(* IEC 61131-3 sources: ics/BLR101_ProenixContact/BLR101_5_ILC171_44/LogicalPOUs/AIO, 3 files *)

(* ---- SensorFB.ST ---- *)
(*@PROPERTIES_EX@
TYPE: POU
LOCALE: 0
IEC_LANGUAGE: ST
PLC_TYPE: independent
PROC_TYPE: independent
GROUP: AIO.FB
*)
(*@KEY@:DESCRIPTION*)

(*@KEY@:END_DESCRIPTION*)
FUNCTION_BLOCK SensorFB

(*Group:Default*)

VAR_IN_OUT
	Snsr_strct :	SNSR;
END_VAR

VAR
	RealValue :	REAL;
	bar_kgf :	REAL;
END_VAR

VAR_IN_OUT
	Buff :	SNSR_BUFF;
END_VAR

VAR
	SumValue :	REAL;
	y :	INT;
	INIT :	BOOL;
	FltrValue :	REAL;
	x :	INT;
END_VAR

VAR_OUTPUT
	Event :	SNSR_EVENT;
END_VAR

VAR_IN_OUT
	Aux_strct :	SNSR_MISC;
END_VAR

VAR_EXTERNAL
	TICK_100MS_PLS :	BOOL;
END_VAR

(*@KEY@: WORKSHEET
NAME: SensorFB
IEC_LANGUAGE: ST
*)

(*================================================================================================*)
(*Fault operation & converting PIW to real value*)
(*================================================================================================*)
IF (Snsr_strct.PIW < 0) OR (Snsr_strct.PIW > Snsr_strct.ADC_Range) OR Snsr_strct.CW.ExtFault OR (Snsr_strct.DiagCode > word#16#8000) THEN		(*Snsr_strct Failed*)
	Snsr_strct.SW.Fault:= TRUE;
	RealValue:= 0.0;
ELSE                                                                    			(*Snsr_strct OK*)
	IF Snsr_strct.ADC_Range <= 0 THEN
		Snsr_strct.ADC_Range:= 1;
	END_IF;
	Snsr_strct.SW.Fault:= FALSE;
	RealValue:= (Snsr_strct.Ymax - Snsr_strct.Ymin) * bar_kgf * INT_TO_REAL(Snsr_strct.PIW) / INT_TO_REAL(Snsr_strct.ADC_Range) + Snsr_strct.Ymin ;
END_IF;

(*================================================================================================*)
(*Converting from bar to kgf/sm2*)
(*================================================================================================*)
IF Snsr_strct.CW.bar_kgf THEN
	bar_kgf:= 1.0197;
ELSE
	bar_kgf:= 1.0;
END_IF;

(*================================================================================================*)
(*SMA filter operation*)
(*================================================================================================*)
if INIT then
	if TICK_100MS_PLS then
		Aux_strct.SamplingTickCount:= Aux_strct.SamplingTickCount + 1;
	end_if;
else
	Aux_strct.SamplingTickCount:= 0;
end_if;

IF Snsr_strct.CW.FltrEn THEN
	IF NOT INIT THEN																(*Initialization*)
		FOR y:= 0 TO 9 DO
			Buff[y]:= RealValue;
			SumValue:= SumValue + Buff[y];
		END_FOR;
		INIT:= TRUE;
	ELSE
		IF Aux_strct.SamplingTickCount >= (Snsr_strct.SamplingTime * 10) THEN		(*Buffer shifting and changing last element*)
			FOR y:= 0 TO 8 DO
				x:= y + 1;
				Buff[y]:= Buff[x];
			END_FOR;
			Buff[9]:= RealValue;
			SumValue:= SumValue + RealValue - Buff[0];
			Aux_strct.SamplingTickCount:= 0;
		END_IF;
		FltrValue:= SumValue / 10.0;
	END_IF;
ELSE
	INIT:= FALSE;
	SumValue:= 0.0;
	FltrValue:= 0.0;
END_IF;

(*================================================================================================*)
(*Snsr_strct output values states*)
(*================================================================================================*)
IF Snsr_strct.CW.SimEn THEN															(*Simulated output value*)
	Snsr_strct.RealValue:= Snsr_strct.SimValue;
ELSIF Snsr_strct.CW.FltrEn THEN														(*Filtered output value*)
	Snsr_strct.RealValue:= FltrValue;
ELSE																				(*Real output value*)
	Snsr_strct.RealValue:= RealValue;
END_IF;

Snsr_strct.IntValue:= REAL_TO_INT(Snsr_strct.RealValue * 100.0);

(*================================================================================================*)
(*Limits operation*)
(*================================================================================================*)
if Snsr_strct.CW.LimEn then
	if (Snsr_strct.RealValue > (Snsr_strct.HH + (Snsr_strct.DeadBand / 2.0))) and not Snsr_strct.SW.HH_alarm  then
		if TICK_100MS_PLS then
			Aux_strct.HHTopDelayCount:= Aux_strct.HHTopDelayCount + 1;
		end_if;
		if Aux_strct.HHTopDelayCount > (Snsr_strct.LimDelay * 10) then
			Snsr_strct.SW.HH_alarm:= true;
		end_if;
	else
		Aux_strct.HHTopDelayCount:= 0;
	end_if;

	if (Snsr_strct.RealValue < (Snsr_strct.HH - (Snsr_strct.DeadBand / 2.0))) and Snsr_strct.SW.HH_alarm then
		if TICK_100MS_PLS then
			Aux_strct.HHBotDelayCount:= Aux_strct.HHBotDelayCount + 1;
		end_if;
		if Aux_strct.HHBotDelayCount > (Snsr_strct.LimDelay * 10) then
			Snsr_strct.SW.HH_alarm:= false;
		end_if;
	else
		Aux_strct.HHBotDelayCount:= 0;
	end_if;

	if (Snsr_strct.RealValue > (Snsr_strct.HL + (Snsr_strct.DeadBand / 2.0))) and not Snsr_strct.SW.HL_alarm then
		if TICK_100MS_PLS then
			Aux_strct.HLTopDelayCount:= Aux_strct.HLTopDelayCount + 1;
		end_if;
		if Aux_strct.HLTopDelayCount > (Snsr_strct.LimDelay * 10) then
			Snsr_strct.SW.HL_alarm:= true;
		end_if;
	else
		Aux_strct.HLTopDelayCount:= 0;
	end_if;

	if (Snsr_strct.RealValue < (Snsr_strct.HL - (Snsr_strct.DeadBand / 2.0))) and Snsr_strct.SW.HL_alarm then
		if TICK_100MS_PLS then
			Aux_strct.HLBotDelayCount:= Aux_strct.HLBotDelayCount + 1;
		end_if;
		if Aux_strct.HLBotDelayCount > (Snsr_strct.LimDelay * 10) then
			Snsr_strct.SW.HL_alarm:= false;
		end_if;
	else
		Aux_strct.HLBotDelayCount:= 0;
	end_if;

	if (Snsr_strct.RealValue < (Snsr_strct.LH - (Snsr_strct.DeadBand / 2.0))) and not Snsr_strct.SW.LH_alarm then
		if TICK_100MS_PLS then
			Aux_strct.LHTopDelayCount:= Aux_strct.LHTopDelayCount + 1;
		end_if;
		if Aux_strct.LHTopDelayCount > (Snsr_strct.LimDelay * 10) then
			Snsr_strct.SW.LH_alarm:= true;
		end_if;
	else
		Aux_strct.LHTopDelayCount:= 0;
	end_if;

	if (Snsr_strct.RealValue > (Snsr_strct.LH + (Snsr_strct.DeadBand / 2.0))) and Snsr_strct.SW.LH_alarm then
		if TICK_100MS_PLS then
			Aux_strct.LHBotDelayCount:= Aux_strct.LHBotDelayCount + 1;
		end_if;
		if Aux_strct.LHBotDelayCount > (Snsr_strct.LimDelay * 10) then
			Snsr_strct.SW.LH_alarm:= false;
		end_if;
	else
		Aux_strct.LHBotDelayCount:= 0;
	end_if;

	if (Snsr_strct.RealValue < (Snsr_strct.LL - (Snsr_strct.DeadBand / 2.0))) and not Snsr_strct.SW.LL_alarm then
		if TICK_100MS_PLS then
			Aux_strct.LLTopDelayCount:= Aux_strct.LLTopDelayCount + 1;
		end_if;
		if Aux_strct.LLTopDelayCount > (Snsr_strct.LimDelay * 10) then
			Snsr_strct.SW.LL_alarm:= true;
		end_if;
	else
		Aux_strct.LLTopDelayCount:= 0;
	end_if;

	if (Snsr_strct.RealValue > (Snsr_strct.LL + (Snsr_strct.DeadBand / 2.0))) and Snsr_strct.SW.LL_alarm then
		if TICK_100MS_PLS then
			Aux_strct.LLBotDelayCount:= Aux_strct.LLBotDelayCount + 1;
		end_if;
		if Aux_strct.LLBotDelayCount > (Snsr_strct.LimDelay * 10) then
			Snsr_strct.SW.LL_alarm:= false;
		end_if;
	else
		Aux_strct.LLBotDelayCount:= 0;
	end_if;

else
	Aux_strct.HHTopDelayCount:= 0;
	Aux_strct.HHBotDelayCount:= 0;

	Aux_strct.HLTopDelayCount:= 0;
	Aux_strct.HLBotDelayCount:= 0;

	Aux_strct.LHTopDelayCount:= 0;
	Aux_strct.LHBotDelayCount:= 0;

	Aux_strct.LLTopDelayCount:= 0;
	Aux_strct.LLBotDelayCount:= 0;

	Snsr_strct.SW.HH_alarm:= FALSE;
	Snsr_strct.SW.HL_alarm:= FALSE;
	Snsr_strct.SW.LH_alarm:= FALSE;
	Snsr_strct.SW.LL_alarm:= FALSE;
end_if;

(*================================================================================================*)
(*Sensor Pulse Events*)
(*================================================================================================*)

Event.Fault:= false;
if Snsr_strct.SW.Fault and not Aux_strct.EVENT_1 then
	Event.Fault:= true;
	Aux_strct.EVENT_1:= true;
elsif not Snsr_strct.SW.Fault then
	Aux_strct.EVENT_1:= false;
end_if;

Event.HH:= false;
if Snsr_strct.SW.HH_alarm and not Aux_strct.EVENT_2 then
	Event.HH:= true;
	Aux_strct.EVENT_2:= true;
elsif not Snsr_strct.SW.HH_alarm then
	Aux_strct.EVENT_2:= false;
end_if;

Event.HL:= false;
if Snsr_strct.SW.HL_alarm and not Aux_strct.EVENT_3 then
	Event.HL:= true;
	Aux_strct.EVENT_3:= true;
elsif not Snsr_strct.SW.HL_alarm then
	Aux_strct.EVENT_3:= false;
end_if;

Event.LH:= false;
if Snsr_strct.SW.LH_alarm and not Aux_strct.EVENT_4 then
	Event.LH:= true;
	Aux_strct.EVENT_4:= true;
elsif not Snsr_strct.SW.LH_alarm then
	Aux_strct.EVENT_4:= false;
end_if;

Event.LL:= false;
if Snsr_strct.SW.LL_alarm and not Aux_strct.EVENT_5 then
	Event.LL:= true;
	Aux_strct.EVENT_5:= true;
elsif not Snsr_strct.SW.LL_alarm then
	Aux_strct.EVENT_5:= false;
end_if;

(*@KEY@: END_WORKSHEET *)
END_FUNCTION_BLOCK

(* ---- AI.ST ---- *)
(*@PROPERTIES_EX@
TYPE: POU
LOCALE: 0
IEC_LANGUAGE: ST
PLC_TYPE: independent
PROC_TYPE: independent
GROUP: AIO
*)
(*@KEY@:DESCRIPTION*)

(*@KEY@:END_DESCRIPTION*)
PROGRAM AI

(*Group:Default*)

VAR_EXTERNAL
	AI :	SENSOR;
END_VAR

VAR
	A07_Param :	IL_AI_4_UI_Para_V1_03;
	i :	INT;
	j :	INT;
	udtA07Param :	ANL_udt_Para_1_5;
	A07_Com :	IL_AI_4_UI_Com_V1_04;
	udtA07Status :	ANL_udt_Status_1_5;
	A07_Ready :	BOOL;
	A07_Err :	BOOL;
	A07_Frmwr :	STRING;
END_VAR

VAR_EXTERNAL
	A07_ProcIn :	ANL_ARR_W_1_4;
	A07_ProcOut :	ANL_ARR_W_1_4;
END_VAR

VAR
	A07_DiagCode :	WORD;
	A07_Diag :	IL_AI_4_UI_Diag_V1_03;
	A08_Param :	IL_AI_4_UI_Para_V1_03;
	udtA08Param :	ANL_udt_Para_1_5;
	A08_Com :	IL_AI_4_UI_Com_V1_04;
	A08_Ready :	BOOL;
	A08_Err :	BOOL;
	A08_DiagCode :	WORD;
	A08_Frmwr :	STRING;
	udtA08Status :	ANL_udt_Status_1_5;
END_VAR

VAR_EXTERNAL
	A08_ProcIn :	ANL_ARR_W_1_4;
	A08_ProcOut :	ANL_ARR_W_1_4;
END_VAR

VAR
	A08_Diag :	IL_AI_4_UI_Diag_V1_03;
	A09_Param :	IL_AI_4_UI_Para_V1_03;
	udtA09Param :	ANL_udt_Para_1_5;
	A09_Com :	IL_AI_4_UI_Com_V1_04;
	A09_Ready :	BOOL;
	A09_Err :	BOOL;
	A09_DiagCode :	WORD;
	A09_Frmwr :	STRING;
	udtA09Status :	ANL_udt_Status_1_5;
END_VAR

VAR_EXTERNAL
	A09_ProcIn :	ANL_ARR_W_1_4;
	A09_ProcOut :	ANL_ARR_W_1_4;
END_VAR

VAR
	A09_Diag :	IL_AI_4_UI_Diag_V1_03;
	A10_Param :	IL_AI_4_UI_Para_V1_03;
	udtA10Param :	ANL_udt_Para_1_5;
	A10_Com :	IL_AI_4_UI_Com_V1_04;
	A10_Ready :	BOOL;
	A10_Err :	BOOL;
	A10_Frmwr :	STRING;
	udtA10Status :	ANL_udt_Status_1_5;
END_VAR

VAR_EXTERNAL
	A10_ProcIn :	ANL_ARR_W_1_4;
	A10_ProcOut :	ANL_ARR_W_1_4;
END_VAR

VAR
	A10_Diag :	IL_AI_4_UI_Diag_V1_03;
	A11_Param :	IL_AI_4_UI_Para_V1_03;
	udtA11Param :	ANL_udt_Para_1_5;
	A11_Com :	IL_AI_4_UI_Com_V1_04;
	A11_Ready :	BOOL;
	A11_Err :	BOOL;
	A11_DiagCode :	WORD;
	A11_Frmwr :	STRING;
	udtA11Status :	ANL_udt_Status_1_5;
END_VAR

VAR_EXTERNAL
	A11_ProcIn :	ANL_ARR_W_1_4;
	A11_ProcOut :	ANL_ARR_W_1_4;
END_VAR

VAR
	A11_Diag :	IL_AI_4_UI_Diag_V1_03;
	A10_DiagCode :	WORD;
	A12_Param :	IL_AI_4_UI_Para_V1_03;
	udtA12Param :	ANL_udt_Para_1_5;
	A12_Com :	IL_AI_4_UI_Com_V1_04;
	A12_Ready :	BOOL;
	A12_Err :	BOOL;
	A12_DiagCode :	WORD;
	A12_Frmwr :	STRING;
	udtA12Status :	ANL_udt_Status_1_5;
END_VAR

VAR_EXTERNAL
	A12_ProcIn :	ANL_ARR_W_1_4;
	A12_ProcOut :	ANL_ARR_W_1_4;
END_VAR

VAR
	A12_Diag :	IL_AI_4_UI_Diag_V1_03;
	SensorsFB :	SensorFB;
	AI_BUFF :	SENSOR_BUFF;
END_VAR

VAR_EXTERNAL
	AI_AUX :	SENSOR_MISC;
	AI_EVENT :	SENSOR_EVENT;
END_VAR

VAR
	A07_Param_2 :	IL_AI_4_UI_Para_V1_03;
	A07_Param_3 :	IL_AI_4_UI_Para_V1_03;
	A07_Param_4 :	IL_AI_4_UI_Para_V1_03;
	REAL_TO_MB :	REAL_TO_MB;
	j1 :	INT;
END_VAR

VAR_EXTERNAL
	MBTCP_Data :	MB_TCP_ARR_W_0_7167;
END_VAR

VAR
	j2 :	INT;
END_VAR

(*@KEY@: WORKSHEET
NAME: AI
IEC_LANGUAGE: ST
*)

(*========================================================================================*)
	(*A07 module parametrization*)
(*========================================================================================*)
for i:= 1 to 4 do
	j:= i - 1;
	A07_Param(iChannel:= i,iMode:= 1,iFilter:= 0,rHighLimit:= int_to_real(AI[j].ADC_Range),rLowLimit:= 0.0,udtPara:= udtA07Param);
	udtA07Param:= A07_Param.udtPara;
end_for;

(*========================================================================================*)
	(*A07 module communication*)
(*========================================================================================*)
A07_Com(xActivate:= true,bSelect:= byte#16#0F,xVoltage:= false,udtPara:=udtA07Param,arrProcIn:= A07_ProcIn);
	A07_Ready			:=	A07_Com.xReady;
	A07_Err				:=	A07_Com.xError;
	A07_DiagCode		:=	A07_Com.wDiagCode;
	A07_Frmwr			:=	A07_Com.strFirmware;
	udtA07Status		:=	A07_Com.udtStatus;
	udtA07Param 		:=	A07_Com.udtPara;
	A07_ProcOut			:=	A07_Com.arrProcOut;
(*========================================================================================*)
	(*A07 module diagnostic*)
(*========================================================================================*)
for i:= 1 to 4 do
	j:= i - 1;
	A07_Diag(udtStatus:= udtA07Status,iChannel:= i);
	AI[j].CW.ExtFault:= not A07_Diag.xDataValid;
	AI[j].DiagCode:= A07_Diag.wDiagCode;
	AI[j].PIW:= real_to_int(A07_Diag.rCurrentValue);
end_for;

(*========================================================================================*)
	(*A08 module parametrization*)
(*========================================================================================*)
for i:= 1 to 4 do
	j:= i + 3;
	A08_Param(iChannel:= i,iMode:= 1,iFilter:= 0,rHighLimit:= int_to_real(AI[j].ADC_Range),rLowLimit:= 0.0,udtPara:= udtA08Param);
	udtA08Param:= A08_Param.udtPara;
end_for;

(*========================================================================================*)
	(*A08 module communication*)
(*========================================================================================*)
A08_Com(xActivate:= true,bSelect:= byte#16#0F,xVoltage:= false,udtPara:=udtA08Param,arrProcIn:= A08_ProcIn);
	A08_Ready			:=	A08_Com.xReady;
	A08_Err				:=	A08_Com.xError;
	A08_DiagCode		:=	A08_Com.wDiagCode;
	A08_Frmwr			:=	A08_Com.strFirmware;
	udtA08Status		:=	A08_Com.udtStatus;
	udtA08Param 		:=	A08_Com.udtPara;
	A08_ProcOut			:=	A08_Com.arrProcOut;
(*========================================================================================*)
	(*A08 module diagnostic*)
(*========================================================================================*)
for i:= 1 to 4 do
	j:= i + 3;
	A08_Diag(udtStatus:= udtA08Status,iChannel:= i);
	AI[j].CW.ExtFault:= not A08_Diag.xDataValid;
	AI[j].DiagCode:= A08_Diag.wDiagCode;
	AI[j].PIW:= real_to_int(A08_Diag.rCurrentValue);
end_for;

(*========================================================================================*)
	(*A09 module parametrization*)
(*========================================================================================*)
for i:= 1 to 4 do
	j:= i + 7;
	A09_Param(iChannel:= i,iMode:= 1,iFilter:= 0,rHighLimit:= int_to_real(AI[j].ADC_Range),rLowLimit:= 0.0,udtPara:= udtA09Param);
	udtA09Param:= A09_Param.udtPara;
end_for;

(*========================================================================================*)
	(*A09 module communication*)
(*========================================================================================*)
A09_Com(xActivate:= true,bSelect:= byte#16#0F,xVoltage:= false,udtPara:=udtA09Param,arrProcIn:= A09_ProcIn);
	A09_Ready			:=	A09_Com.xReady;
	A09_Err				:=	A09_Com.xError;
	A09_DiagCode		:=	A09_Com.wDiagCode;
	A09_Frmwr			:=	A09_Com.strFirmware;
	udtA09Status		:=	A09_Com.udtStatus;
	udtA09Param 		:=	A09_Com.udtPara;
	A09_ProcOut			:=	A09_Com.arrProcOut;
(*========================================================================================*)
	(*A09 module diagnostic*)
(*========================================================================================*)
for i:= 1 to 4 do
	j:= i + 7;
	A09_Diag(udtStatus:= udtA09Status,iChannel:= i);
	AI[j].CW.ExtFault:= not A09_Diag.xDataValid;
	AI[j].DiagCode:= A09_Diag.wDiagCode;
	AI[j].PIW:= real_to_int(A09_Diag.rCurrentValue);
end_for;

(*========================================================================================*)
	(*A10 module parametrization*)
(*========================================================================================*)
	A10_Param(iChannel:= 1,iMode:= 1,iFilter:= 0,rHighLimit:= int_to_real(AI[12].ADC_Range),rLowLimit:= 0.0,udtPara:= udtA10Param);
	udtA10Param:= A10_Param.udtPara;

(*========================================================================================*)
	(*A10 module communication*)
(*========================================================================================*)
A10_Com(xActivate:= true,bSelect:= byte#16#01,xVoltage:= false,udtPara:=udtA10Param,arrProcIn:= A10_ProcIn);
	A10_Ready			:=	A10_Com.xReady;
	A10_Err				:=	A10_Com.xError;
	A10_DiagCode		:=	A10_Com.wDiagCode;
	A10_Frmwr			:=	A10_Com.strFirmware;
	udtA10Status		:=	A10_Com.udtStatus;
	udtA10Param 		:=	A10_Com.udtPara;
	A10_ProcOut			:=	A10_Com.arrProcOut;
(*========================================================================================*)
	(*A10 module diagnostic*)
(*========================================================================================*)
	A10_Diag(udtStatus:= udtA10Status,iChannel:= 1);
	AI[12].CW.ExtFault:= not A10_Diag.xDataValid;
	AI[12].DiagCode:= A10_Diag.wDiagCode;
	AI[12].PIW:= real_to_int(A10_Diag.rCurrentValue);

(*========================================================================================*)
	(*A11 module parametrization*)
(*========================================================================================*)
for i:= 1 to 3 do
	j:= i + 15;
	A11_Param(iChannel:= i,iMode:= 0,iFilter:= 0,rHighLimit:= 10000.0,rLowLimit:= 0.0,udtPara:= udtA11Param);
	udtA11Param:= A11_Param.udtPara;
end_for;

(*========================================================================================*)
	(*A11 module communication*)
(*========================================================================================*)
A11_Com(xActivate:= true,bSelect:= byte#16#07,xVoltage:= false,udtPara:=udtA11Param,arrProcIn:= A11_ProcIn);
	A11_Ready			:=	A11_Com.xReady;
	A11_Err				:=	A11_Com.xError;
	A11_DiagCode		:=	A11_Com.wDiagCode;
	A11_Frmwr			:=	A11_Com.strFirmware;
	udtA11Status		:=	A11_Com.udtStatus;
	udtA11Param 		:=	A11_Com.udtPara;
	A11_ProcOut			:=	A11_Com.arrProcOut;
(*========================================================================================*)
	(*A11 module diagnostic*)
(*========================================================================================*)
for i:= 1 to 3 do
	j:= i + 15;
	A11_Diag(udtStatus:= udtA11Status,iChannel:= i);
	AI[j].CW.ExtFault:= not A11_Diag.xDataValid;
	AI[j].DiagCode:= A11_Diag.wDiagCode;
	AI[j].PIW:= real_to_int(A11_Diag.rCurrentValue);
end_for;

(*========================================================================================*)
	(*A12 module parametrization*)
(*========================================================================================*)
for i:= 1 to 2 do
	j:= i + 19;
	A12_Param(iChannel:= i,iMode:= 0,iFilter:= 0,rHighLimit:= 10000.0,rLowLimit:= 0.0,udtPara:= udtA12Param);
	udtA12Param:= A12_Param.udtPara;
end_for;

(*========================================================================================*)
	(*A12 module communication*)
(*========================================================================================*)
A12_Com(xActivate:= true,bSelect:= byte#16#03,xVoltage:= false,udtPara:=udtA12Param,arrProcIn:= A12_ProcIn);
	A12_Ready			:=	A12_Com.xReady;
	A12_Err				:=	A12_Com.xError;
	A12_DiagCode		:=	A12_Com.wDiagCode;
	A12_Frmwr			:=	A12_Com.strFirmware;
	udtA12Status		:=	A12_Com.udtStatus;
	udtA12Param 		:=	A12_Com.udtPara;
	A12_ProcOut			:=	A12_Com.arrProcOut;
(*========================================================================================*)
	(*A12 module diagnostic*)
(*========================================================================================*)
for i:= 1 to 2 do
	j:= i + 19;
	A12_Diag(udtStatus:= udtA12Status,iChannel:= i);
	AI[j].CW.ExtFault:= not A12_Diag.xDataValid;
	AI[j].DiagCode:= A12_Diag.wDiagCode;
	AI[j].PIW:= real_to_int(A12_Diag.rCurrentValue);
end_for;

(*================================================================================================*)
	(*FC AO param*)
(*================================================================================================*)
for i:= 16 to 18 do
	j:= i * 32 + 104;
	j1:= j + 1;
	j2:= j + 2;

	REAL_TO_MB(IN:=100.0);
	MBTCP_Data[j]:=REAL_TO_MB.LoWord;
	MBTCP_Data[j1]:=REAL_TO_MB.HiWord;

	MBTCP_Data[j2]:= word#10000;
end_for;

for i:= 20 to 21 do
	j:= i * 32 + 104;
	j1:= j + 1;
	j2:= j + 2;

	REAL_TO_MB(IN:=100.0);
	MBTCP_Data[j]:=REAL_TO_MB.LoWord;
	MBTCP_Data[j1]:=REAL_TO_MB.HiWord;

	MBTCP_Data[j2]:= word#10000;
end_for;

(*================================================================================================*)
	(*Analog sensors processing*)
(*================================================================================================*)

AI[0].CW.bar_kgf:= true;
for i:= 2 to 12 do
	AI[i].CW.bar_kgf:= true;
end_for;

for i:= 0 to 23 do
	SensorsFB(Snsr_strct:= AI[i],Buff:= AI_Buff[i],Aux_strct:= AI_AUX[i]);
	AI[i]:=SensorsFB.Snsr_strct;
	AI_BUFF[i]:=SensorsFB.Buff;
	AI_EVENT[i]:=SensorsFB.Event;
	AI_AUX[i]:=SensorsFB.Aux_strct;
end_for;

(*@KEY@: END_WORKSHEET *)
END_PROGRAM

(* ---- AO.ST ---- *)
(*@PROPERTIES_EX@
TYPE: POU
LOCALE: 0
IEC_LANGUAGE: ST
PLC_TYPE: independent
PROC_TYPE: independent
GROUP: AIO
*)
(*@KEY@:DESCRIPTION*)

(*@KEY@:END_DESCRIPTION*)
PROGRAM AO

(*Group:Default*)

VAR
	i :	INT;
	A13_Param :	IL_AO_2_UI_Para_V1_02;
	j :	INT;
END_VAR

VAR_EXTERNAL
	M_AUX :	MOTOR_MISC;
END_VAR

VAR
	arrParamA13 :	ANL_ARR_Para_1_2;
	A13_Com :	IL_AO_2_UI_V1_02;
	A13_Ready :	BOOL;
	A13_Err :	BOOL;
	A13_DiagCode :	WORD;
	A13_AddDiagCode :	WORD;
	A13_arrDiag :	ANL_ARR_Diag_1_2;
END_VAR

VAR_EXTERNAL
	A13_ProcIn :	ANL_ARR_W_1_4;
	A13_ProcOut :	ANL_ARR_W_1_4;
END_VAR

VAR
	A13_CH1_Diag :	IL_AO_2_UI_Diag_V1_01;
	A13_CH2_Diag :	IL_AO_2_UI_Diag_V1_01;
	A13_CH1_Err :	BOOL;
	A13_CH1_ErrCode :	WORD;
	A13_CH2_Err :	BOOL;
	A13_CH2_ErrCode :	WORD;
	A14_Param :	IL_AO_2_UI_Para_V1_02;
	arrParamA14 :	ANL_ARR_Para_1_2;
	A14_Com :	IL_AO_2_UI_V1_02;
	A14_Ready :	BOOL;
	A14_Err :	BOOL;
	A14_DiagCode :	WORD;
	A14_AddDiagCode :	WORD;
	A14_arrDiag :	ANL_ARR_Diag_1_2;
END_VAR

VAR_EXTERNAL
	A14_ProcIn :	ANL_ARR_W_1_4;
	A14_ProcOut :	ANL_ARR_W_1_4;
END_VAR

VAR
	A14_CH1_Diag :	IL_AO_2_UI_Diag_V1_01;
	A14_CH1_Err :	BOOL;
	A14_CH1_ErrCode :	WORD;
	A16_Param :	IL_AO_2_UI_Para_V1_02;
	arrParamA16 :	ANL_ARR_Para_1_2;
	A16_Com :	IL_AO_2_UI_V1_02;
	A16_Ready :	BOOL;
	A16_Err :	BOOL;
	A16_DiagCode :	WORD;
	A16_AddDiagCode :	WORD;
	A16_arrDiag :	ANL_ARR_Diag_1_2;
END_VAR

VAR_EXTERNAL
	A16_ProcIn :	ANL_ARR_W_1_4;
	A16_ProcOut :	ANL_ARR_W_1_4;
END_VAR

VAR
	A16_CH1_Diag :	IL_AO_2_UI_Diag_V1_01;
	A16_CH1_Err :	BOOL;
	A16_CH1_ErrCode :	WORD;
	A16_CH2_Diag :	IL_AO_2_UI_Diag_V1_01;
	A16_CH2_Err :	BOOL;
	A16_CH2_ErrCode :	WORD;
END_VAR

(*@KEY@: WORKSHEET
NAME: AO
IEC_LANGUAGE: ST
*)
(*========================================================================================*)
	(*A13 module parametrization*)
(*========================================================================================*)
for i:= 1 to 2 do
	j:= i - 1;
	A13_Param(iChannelNo:= i,iRange:= 2,rHiLim:= 50.0,rLoLim:= 0.0,rSetValue:= M_AUX[j].SetValue,arrParameter:= arrParamA13);
	arrParamA13:= A13_Param.arrParameter;
end_for;

(*========================================================================================*)
	(*A13 module communication*)
(*========================================================================================*)
A13_Com(xActivate:= true,iSelectCH:= 3,arrParameter:= arrParamA13,arrProcIN:= A13_ProcIn);
	A13_Ready			:=	A13_Com.xReady;
	A13_Err				:=	A13_Com.xError;
	A13_DiagCode		:=	A13_Com.wDiagCode;
	A13_AddDiagCode		:=	A13_Com.wAddDiagCode;
	A13_arrDiag			:=	A13_Com.arrDiag;
	A13_ProcOut			:=	A13_Com.arrProcOUT;

(*========================================================================================*)
	(*A13 module diagnostic*)
(*========================================================================================*)
A13_CH1_Diag(iChannelNo:= 1,arrDiag:=A13_arrDiag);
A13_CH1_Err				:=	A13_CH1_Diag.xError;
A13_CH1_ErrCode			:=	A13_CH1_Diag.wErrorCode;
A13_arrDiag				:=	A13_CH1_Diag.arrDiag;

A13_CH2_Diag(iChannelNo:= 2,arrDiag:=A13_arrDiag);
A13_CH2_Err				:=	A13_CH2_Diag.xError;
A13_CH2_ErrCode			:=	A13_CH2_Diag.wErrorCode;
A13_arrDiag				:=	A13_CH2_Diag.arrDiag;

(*========================================================================================*)
	(*A14 module parametrization*)
(*========================================================================================*)
A14_Param(iChannelNo:= 1,iRange:= 2,rHiLim:= 50.0,rLoLim:= 0.0,rSetValue:= M_AUX[2].SetValue,arrParameter:= arrParamA14);
	arrParamA14:= A14_Param.arrParameter;

(*========================================================================================*)
	(*A14 module communication*)
(*========================================================================================*)
A14_Com(xActivate:= true,iSelectCH:= 1,arrParameter:= arrParamA14,arrProcIN:= A14_ProcIn);
	A14_Ready			:=	A14_Com.xReady;
	A14_Err				:=	A14_Com.xError;
	A14_DiagCode		:=	A14_Com.wDiagCode;
	A14_AddDiagCode		:=	A14_Com.wAddDiagCode;
	A14_arrDiag			:=	A14_Com.arrDiag;
	A14_ProcOut			:=	A14_Com.arrProcOUT;

(*========================================================================================*)
	(*A14 module diagnostic*)
(*========================================================================================*)
A14_CH1_Diag(iChannelNo:= 1,arrDiag:=A14_arrDiag);
A14_CH1_Err				:=	A14_CH1_Diag.xError;
A14_CH1_ErrCode			:=	A14_CH1_Diag.wErrorCode;
A14_arrDiag				:=	A14_CH1_Diag.arrDiag;

(*========================================================================================*)
	(*A16 module parametrization*)
(*========================================================================================*)
for i:= 1 to 2 do
	j:= i + 2;
	A16_Param(iChannelNo:= i,iRange:= 2,rHiLim:= 50.0,rLoLim:= 0.0,rSetValue:= M_AUX[j].SetValue,arrParameter:= arrParamA16);
	arrParamA16:= A16_Param.arrParameter;
end_for;

(*========================================================================================*)
	(*A16 module communication*)
(*========================================================================================*)
A16_Com(xActivate:= true,iSelectCH:= 3,arrParameter:= arrParamA16,arrProcIN:= A16_ProcIn);
	A16_Ready			:=	A16_Com.xReady;
	A16_Err				:=	A16_Com.xError;
	A16_DiagCode		:=	A16_Com.wDiagCode;
	A16_AddDiagCode		:=	A16_Com.wAddDiagCode;
	A16_arrDiag			:=	A16_Com.arrDiag;
	A16_ProcOut			:=	A16_Com.arrProcOUT;

(*========================================================================================*)
	(*A16 module diagnostic*)
(*========================================================================================*)
A16_CH1_Diag(iChannelNo:= 1,arrDiag:=A16_arrDiag);
A16_CH1_Err				:=	A16_CH1_Diag.xError;
A16_CH1_ErrCode			:=	A16_CH1_Diag.wErrorCode;
A16_arrDiag				:=	A16_CH1_Diag.arrDiag;

A16_CH2_Diag(iChannelNo:= 2,arrDiag:=A16_arrDiag);
A16_CH2_Err				:=	A16_CH2_Diag.xError;
A16_CH2_ErrCode			:=	A16_CH2_Diag.wErrorCode;
A16_arrDiag				:=	A16_CH2_Diag.arrDiag;

(*@KEY@: END_WORKSHEET *)
END_PROGRAM
